(* Schneider Machine Expert - Basic project XIC-XIO parallel neg-coil, file version 1.6.0.0 *)
(* ProjectInformations: Name=New project *)

HARDWARE
  Cpu 0: TM221CE16R
  EthernetConfiguration: NetworkName=M221, IpAllocationMode=FixedAddress, IpAddress=0.0.0.0, SubnetMask=0.0.0.0
  SerialLineConfiguration: Baud=Baud19200, Parity=ParityEven, DataBits=DataBits8, StopBits=StopBits1, PhysicalMedium=PhysicalMediumRs485, TransmissionMode=TransmissionModeModbusRtu, SlaveId=1, Addressing=SlaveAddressing
  MastTask: UsePeriodScanMode=false, PeriodScan=100
  FastTask: Period=255
  CpuBehavior: StartingMode=StartAsPreviousState, AutoSaveRamOnEeprom=true, WatchdogPeriod=250

SYMBOLS  (address, symbol, comment, settings)

POU New POU
  (* SectionNumber=1 *)

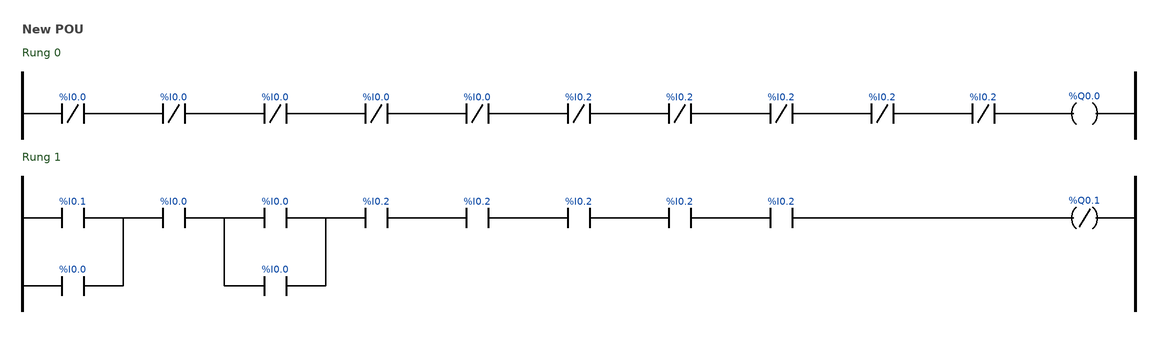

// Rung 0
  LDN %I0.0
  ANDN %I0.0
  ANDN %I0.0
  ANDN %I0.0
  ANDN %I0.0
  ANDN %I0.2
  ANDN %I0.2
  ANDN %I0.2
  ANDN %I0.2
  ANDN %I0.2
  ST %Q0.0
  // as ST:
  //   %Q0.0 := NOT %I0.0 AND NOT %I0.0 AND NOT %I0.0 AND NOT %I0.0 AND NOT %I0.0 AND NOT %I0.2 AND NOT %I0.2 AND NOT %I0.2 AND NOT %I0.2 AND NOT %I0.2;

// Rung 1
  LD %I0.1
  OR %I0.0
  AND %I0.0
  AND( %I0.0
  OR %I0.0
  )
  AND %I0.2
  AND %I0.2
  AND %I0.2
  AND %I0.2
  AND %I0.2
  STN %Q0.1
  // as ST:
  //   %Q0.1 := NOT ((%I0.1 OR %I0.0) AND %I0.0 AND (%I0.0 OR %I0.0) AND %I0.2 AND %I0.2 AND %I0.2 AND %I0.2 AND %I0.2);
